FUNCTION F_CHARTOBYTE : BYTE
VAR_INPUT
	Char : T_Char;
END_VAR

F_CHARTOBYTE := Char[0];

END_FUNCTION

(* stored: Version 1.1.0.1, ProductVersion 3.1.4024.4
   POU F_CHARTOBYTE: Id {ffe05fa9-9469-43fe-addd-9fa01c298718}, SpecialFunc None *)
